{attribute 'qualified_only'}
VAR_GLOBAL
	fEncoderDia 	: LREAL := 0.0443; 	// [m]
	fEncoderBit 	: LREAL := 65536.0; // [Bit/turn]
	fEncoderDist	: LREAL := fEncoderDia * Tc2_System.Global_Variables.PI; // [m]
END_VAR

(* stored: Version 1.1.0.1
   GVL G_Winch: Id {8f44b33e-e33f-4c04-b80f-3076fdbd6d35} *)
